(* CODESYS project festo_tcmc3.library
   Company: Festo AG & Co. KG
   DefaultNamespace: Festo_TcMC3
   Version: 3.1.1
   Placeholder: Festo TcMC Library for TwinCAT 3
   Author: Festo AG & Co. KG
   Title: Festo TcMC Library for TwinCAT 3
   Description: Additional Function blocks 
      to use Festo CMMx-xx Controller 
      with Beckhoff TwinCAT NC Environment

Project tree, tasks and I/O mapping:
  libraries: Tc2_EtherCAT, * (Beckhoff Automation GmbH); Tc2_Math, * (Beckhoff Automation GmbH); Tc2_MC2, * (Beckhoff Automation GmbH); Tc2_NC, * (Beckhoff Automation GmbH); Tc2_Standard, * (Beckhoff Automation GmbH); Tc2_System, * (Beckhoff Automation GmbH); Tc2_Utilities, * (Beckhoff Automation GmbH)
  Data types/
    data type EFesto_CAN_IDX
    data type EFesto_CAN_SUB_IDX
  POUs/
    function block Festo_GetDriveError [ST]
    function block Festo_MC_Home [ST]
    function block Festo_ReadCanObj [ST]
    function block Festo_WriteCanObj [ST]
  Version/
    global variables Global_Version
  Visualizations/
*)

// Data types/EFesto_CAN_IDX
TYPE EFesto_CAN_IDX :
(
	E_FESTO_CAN_IDX_NONE			:= 16#0,
	E_FESTO_CAN_IDX_ERROR			:= 16#1003

);
END_TYPE

// Data types/EFesto_CAN_SUB_IDX
TYPE EFesto_CAN_SUB_IDX :
(
	E_FESTO_CAN_IDX_SUB_00			:= 16#0,
	E_FESTO_CAN_IDX_SUB_01			:= 16#1,
	E_FESTO_CAN_IDX_SUB_02			:= 16#2,
	E_FESTO_CAN_IDX_SUB_03			:= 16#3,
	E_FESTO_CAN_IDX_SUB_04			:= 16#4,
	E_FESTO_CAN_IDX_SUB_05			:= 16#5,
	E_FESTO_CAN_IDX_SUB_06			:= 16#6,
	E_FESTO_CAN_IDX_SUB_07			:= 16#7,
	E_FESTO_CAN_IDX_SUB_08			:= 16#8,
	E_FESTO_CAN_IDX_SUB_09			:= 16#9,
	E_FESTO_CAN_IDX_SUB_0A			:= 16#0A,
	E_FESTO_CAN_IDX_SUB_0B			:= 16#0B,
	E_FESTO_CAN_IDX_SUB_0C			:= 16#0C,
	E_FESTO_CAN_IDX_SUB_0D			:= 16#0D,
	E_FESTO_CAN_IDX_SUB_0E			:= 16#0E,
	E_FESTO_CAN_IDX_SUB_0F			:= 16#0F,
	E_FESTO_CAN_IDX_SUB_10			:= 16#10,
	E_FESTO_CAN_IDX_SUB_11			:= 16#11,
	E_FESTO_CAN_IDX_SUB_12			:= 16#12,
	E_FESTO_CAN_IDX_SUB_13			:= 16#13,
	E_FESTO_CAN_IDX_SUB_14			:= 16#14,
	E_FESTO_CAN_IDX_SUB_15			:= 16#15,
	E_FESTO_CAN_IDX_SUB_16			:= 16#16,
	E_FESTO_CAN_IDX_SUB_17			:= 16#17,
	E_FESTO_CAN_IDX_SUB_18			:= 16#18,
	E_FESTO_CAN_IDX_SUB_19			:= 16#19,
	E_FESTO_CAN_IDX_SUB_1A			:= 16#1A,
	E_FESTO_CAN_IDX_SUB_1B			:= 16#1B,
	E_FESTO_CAN_IDX_SUB_1C			:= 16#1C,
	E_FESTO_CAN_IDX_SUB_1D			:= 16#1D,
	E_FESTO_CAN_IDX_SUB_1E			:= 16#1E,
	E_FESTO_CAN_IDX_SUB_1F			:= 16#1F,
	E_FESTO_CAN_IDX_SUB_20			:= 16#20,
	E_FESTO_CAN_IDX_SUB_21			:= 16#21,
	E_FESTO_CAN_IDX_SUB_22			:= 16#22,
	E_FESTO_CAN_IDX_SUB_23			:= 16#23,
	E_FESTO_CAN_IDX_SUB_24			:= 16#24,
	E_FESTO_CAN_IDX_SUB_25			:= 16#25,
	E_FESTO_CAN_IDX_SUB_26			:= 16#26,
	E_FESTO_CAN_IDX_SUB_27			:= 16#27,
	E_FESTO_CAN_IDX_SUB_28			:= 16#28,
	E_FESTO_CAN_IDX_SUB_29			:= 16#29,
	E_FESTO_CAN_IDX_SUB_2A			:= 16#2A,
	E_FESTO_CAN_IDX_SUB_2B			:= 16#2B,
	E_FESTO_CAN_IDX_SUB_2C			:= 16#2C,
	E_FESTO_CAN_IDX_SUB_2D			:= 16#2D,
	E_FESTO_CAN_IDX_SUB_2E			:= 16#2E,
	E_FESTO_CAN_IDX_SUB_2F			:= 16#2F,
	E_FESTO_CAN_IDX_SUB_30			:= 16#30,
	E_FESTO_CAN_IDX_SUB_31			:= 16#31,
	E_FESTO_CAN_IDX_SUB_32			:= 16#32,
	E_FESTO_CAN_IDX_SUB_33			:= 16#33,
	E_FESTO_CAN_IDX_SUB_34			:= 16#34,
	E_FESTO_CAN_IDX_SUB_35			:= 16#35,
	E_FESTO_CAN_IDX_SUB_36			:= 16#36,
	E_FESTO_CAN_IDX_SUB_37			:= 16#37,
	E_FESTO_CAN_IDX_SUB_38			:= 16#38,
	E_FESTO_CAN_IDX_SUB_39			:= 16#39,
	E_FESTO_CAN_IDX_SUB_3A			:= 16#3A,
	E_FESTO_CAN_IDX_SUB_3B			:= 16#3B,
	E_FESTO_CAN_IDX_SUB_3C			:= 16#3C,
	E_FESTO_CAN_IDX_SUB_3D			:= 16#3D,
	E_FESTO_CAN_IDX_SUB_3E			:= 16#3E,
	E_FESTO_CAN_IDX_SUB_3F			:= 16#3F,
	E_FESTO_CAN_IDX_SUB_40			:= 16#40,
	E_FESTO_CAN_IDX_SUB_41			:= 16#41,
	E_FESTO_CAN_IDX_SUB_42			:= 16#42,
	E_FESTO_CAN_IDX_SUB_43			:= 16#43,
	E_FESTO_CAN_IDX_SUB_44			:= 16#44,
	E_FESTO_CAN_IDX_SUB_45			:= 16#45,
	E_FESTO_CAN_IDX_SUB_46			:= 16#46,
	E_FESTO_CAN_IDX_SUB_47			:= 16#47,
	E_FESTO_CAN_IDX_SUB_48			:= 16#48,
	E_FESTO_CAN_IDX_SUB_49			:= 16#49,
	E_FESTO_CAN_IDX_SUB_4A			:= 16#4A,
	E_FESTO_CAN_IDX_SUB_4B			:= 16#4B,
	E_FESTO_CAN_IDX_SUB_4C			:= 16#4C,
	E_FESTO_CAN_IDX_SUB_4D			:= 16#4D,
	E_FESTO_CAN_IDX_SUB_4E			:= 16#4E,
	E_FESTO_CAN_IDX_SUB_4F			:= 16#4F,
	E_FESTO_CAN_IDX_SUB_50			:= 16#50,
	E_FESTO_CAN_IDX_SUB_51			:= 16#51,
	E_FESTO_CAN_IDX_SUB_52			:= 16#52,
	E_FESTO_CAN_IDX_SUB_53			:= 16#53,
	E_FESTO_CAN_IDX_SUB_54			:= 16#54,
	E_FESTO_CAN_IDX_SUB_55			:= 16#55,
	E_FESTO_CAN_IDX_SUB_56			:= 16#56,
	E_FESTO_CAN_IDX_SUB_57			:= 16#57,
	E_FESTO_CAN_IDX_SUB_58			:= 16#58,
	E_FESTO_CAN_IDX_SUB_59			:= 16#59,
	E_FESTO_CAN_IDX_SUB_5A			:= 16#5A,
	E_FESTO_CAN_IDX_SUB_5B			:= 16#5B,
	E_FESTO_CAN_IDX_SUB_5C			:= 16#5C,
	E_FESTO_CAN_IDX_SUB_5D			:= 16#5D,
	E_FESTO_CAN_IDX_SUB_5E			:= 16#5E,
	E_FESTO_CAN_IDX_SUB_5F			:= 16#5F,
	E_FESTO_CAN_IDX_SUB_60			:= 16#60,
	E_FESTO_CAN_IDX_SUB_61			:= 16#61,
	E_FESTO_CAN_IDX_SUB_62			:= 16#62,
	E_FESTO_CAN_IDX_SUB_63			:= 16#63,
	E_FESTO_CAN_IDX_SUB_64			:= 16#64,
	E_FESTO_CAN_IDX_SUB_65			:= 16#65,
	E_FESTO_CAN_IDX_SUB_66			:= 16#66,
	E_FESTO_CAN_IDX_SUB_67			:= 16#67,
	E_FESTO_CAN_IDX_SUB_68			:= 16#68,
	E_FESTO_CAN_IDX_SUB_69			:= 16#69,
	E_FESTO_CAN_IDX_SUB_6A			:= 16#6A,
	E_FESTO_CAN_IDX_SUB_6B			:= 16#6B,
	E_FESTO_CAN_IDX_SUB_6C			:= 16#6C,
	E_FESTO_CAN_IDX_SUB_6D			:= 16#6D,
	E_FESTO_CAN_IDX_SUB_6E			:= 16#6E,
	E_FESTO_CAN_IDX_SUB_6F			:= 16#6F,
	E_FESTO_CAN_IDX_SUB_70			:= 16#70,
	E_FESTO_CAN_IDX_SUB_71			:= 16#71,
	E_FESTO_CAN_IDX_SUB_72			:= 16#72,
	E_FESTO_CAN_IDX_SUB_73			:= 16#73,
	E_FESTO_CAN_IDX_SUB_74			:= 16#74,
	E_FESTO_CAN_IDX_SUB_75			:= 16#75,
	E_FESTO_CAN_IDX_SUB_76			:= 16#76,
	E_FESTO_CAN_IDX_SUB_77			:= 16#77,
	E_FESTO_CAN_IDX_SUB_78			:= 16#78,
	E_FESTO_CAN_IDX_SUB_79			:= 16#79,
	E_FESTO_CAN_IDX_SUB_7A			:= 16#7A,
	E_FESTO_CAN_IDX_SUB_7B			:= 16#7B,
	E_FESTO_CAN_IDX_SUB_7C			:= 16#7C,
	E_FESTO_CAN_IDX_SUB_7D			:= 16#7D,
	E_FESTO_CAN_IDX_SUB_7E			:= 16#7E,
	E_FESTO_CAN_IDX_SUB_7F			:= 16#7F,
	E_FESTO_CAN_IDX_SUB_80			:= 16#80,
	E_FESTO_CAN_IDX_SUB_81			:= 16#81,
	E_FESTO_CAN_IDX_SUB_82			:= 16#82,
	E_FESTO_CAN_IDX_SUB_83			:= 16#83,
	E_FESTO_CAN_IDX_SUB_84			:= 16#84,
	E_FESTO_CAN_IDX_SUB_85			:= 16#85,
	E_FESTO_CAN_IDX_SUB_86			:= 16#86,
	E_FESTO_CAN_IDX_SUB_87			:= 16#87,
	E_FESTO_CAN_IDX_SUB_88			:= 16#88,
	E_FESTO_CAN_IDX_SUB_89			:= 16#89,
	E_FESTO_CAN_IDX_SUB_8A			:= 16#8A,
	E_FESTO_CAN_IDX_SUB_8B			:= 16#8B,
	E_FESTO_CAN_IDX_SUB_8C			:= 16#8C,
	E_FESTO_CAN_IDX_SUB_8D			:= 16#8D,
	E_FESTO_CAN_IDX_SUB_8E			:= 16#8E,
	E_FESTO_CAN_IDX_SUB_8F			:= 16#8F,
	E_FESTO_CAN_IDX_SUB_90			:= 16#90,
	E_FESTO_CAN_IDX_SUB_91			:= 16#91,
	E_FESTO_CAN_IDX_SUB_92			:= 16#92,
	E_FESTO_CAN_IDX_SUB_93			:= 16#93,
	E_FESTO_CAN_IDX_SUB_94			:= 16#94,
	E_FESTO_CAN_IDX_SUB_95			:= 16#95,
	E_FESTO_CAN_IDX_SUB_96			:= 16#96,
	E_FESTO_CAN_IDX_SUB_97			:= 16#97,
	E_FESTO_CAN_IDX_SUB_98			:= 16#98,
	E_FESTO_CAN_IDX_SUB_99			:= 16#99,
	E_FESTO_CAN_IDX_SUB_9A			:= 16#9A,
	E_FESTO_CAN_IDX_SUB_9B			:= 16#9B,
	E_FESTO_CAN_IDX_SUB_9C			:= 16#9C,
	E_FESTO_CAN_IDX_SUB_9D			:= 16#9D,
	E_FESTO_CAN_IDX_SUB_9E			:= 16#9E,
	E_FESTO_CAN_IDX_SUB_9F			:= 16#9F,
	E_FESTO_CAN_IDX_SUB_A0			:= 16#A0,
	E_FESTO_CAN_IDX_SUB_A1			:= 16#A1,
	E_FESTO_CAN_IDX_SUB_A2			:= 16#A2,
	E_FESTO_CAN_IDX_SUB_A3			:= 16#A3,
	E_FESTO_CAN_IDX_SUB_A4			:= 16#A4,
	E_FESTO_CAN_IDX_SUB_A5			:= 16#A5,
	E_FESTO_CAN_IDX_SUB_A6			:= 16#A6,
	E_FESTO_CAN_IDX_SUB_A7			:= 16#A7,
	E_FESTO_CAN_IDX_SUB_A8			:= 16#A8,
	E_FESTO_CAN_IDX_SUB_A9			:= 16#A9,
	E_FESTO_CAN_IDX_SUB_AA			:= 16#AA,
	E_FESTO_CAN_IDX_SUB_AB			:= 16#AB,
	E_FESTO_CAN_IDX_SUB_AC			:= 16#AC,
	E_FESTO_CAN_IDX_SUB_AD			:= 16#AD,
	E_FESTO_CAN_IDX_SUB_AE			:= 16#AE,
	E_FESTO_CAN_IDX_SUB_AF			:= 16#AF,
	E_FESTO_CAN_IDX_SUB_B0			:= 16#B0,
	E_FESTO_CAN_IDX_SUB_B1			:= 16#B1,
	E_FESTO_CAN_IDX_SUB_B2			:= 16#B2,
	E_FESTO_CAN_IDX_SUB_B3			:= 16#B3,
	E_FESTO_CAN_IDX_SUB_B4			:= 16#B4,
	E_FESTO_CAN_IDX_SUB_B5			:= 16#B5,
	E_FESTO_CAN_IDX_SUB_B6			:= 16#B6,
	E_FESTO_CAN_IDX_SUB_B7			:= 16#B7,
	E_FESTO_CAN_IDX_SUB_B8			:= 16#B8,
	E_FESTO_CAN_IDX_SUB_B9			:= 16#B9,
	E_FESTO_CAN_IDX_SUB_BA			:= 16#BA,
	E_FESTO_CAN_IDX_SUB_BB			:= 16#BB,
	E_FESTO_CAN_IDX_SUB_BC			:= 16#BC,
	E_FESTO_CAN_IDX_SUB_BD			:= 16#BD,
	E_FESTO_CAN_IDX_SUB_BE			:= 16#BE,
	E_FESTO_CAN_IDX_SUB_BF			:= 16#BF,
	E_FESTO_CAN_IDX_SUB_C0			:= 16#C0,
	E_FESTO_CAN_IDX_SUB_C1			:= 16#C1,
	E_FESTO_CAN_IDX_SUB_C2			:= 16#C2,
	E_FESTO_CAN_IDX_SUB_C3			:= 16#C3,
	E_FESTO_CAN_IDX_SUB_C4			:= 16#C4,
	E_FESTO_CAN_IDX_SUB_C5			:= 16#C5,
	E_FESTO_CAN_IDX_SUB_C6			:= 16#C6,
	E_FESTO_CAN_IDX_SUB_C7			:= 16#C7,
	E_FESTO_CAN_IDX_SUB_C8			:= 16#C8,
	E_FESTO_CAN_IDX_SUB_C9			:= 16#C9,
	E_FESTO_CAN_IDX_SUB_CA			:= 16#CA,
	E_FESTO_CAN_IDX_SUB_CB			:= 16#CB,
	E_FESTO_CAN_IDX_SUB_CC			:= 16#CC,
	E_FESTO_CAN_IDX_SUB_CD			:= 16#CD,
	E_FESTO_CAN_IDX_SUB_CE			:= 16#CE,
	E_FESTO_CAN_IDX_SUB_CF			:= 16#CF,
	E_FESTO_CAN_IDX_SUB_D0			:= 16#D0,
	E_FESTO_CAN_IDX_SUB_D1			:= 16#D1,
	E_FESTO_CAN_IDX_SUB_D2			:= 16#D2,
	E_FESTO_CAN_IDX_SUB_D3			:= 16#D3,
	E_FESTO_CAN_IDX_SUB_D4			:= 16#D4,
	E_FESTO_CAN_IDX_SUB_D5			:= 16#D5,
	E_FESTO_CAN_IDX_SUB_D6			:= 16#D6,
	E_FESTO_CAN_IDX_SUB_D7			:= 16#D7,
	E_FESTO_CAN_IDX_SUB_D8			:= 16#D8,
	E_FESTO_CAN_IDX_SUB_D9			:= 16#D9,
	E_FESTO_CAN_IDX_SUB_DA			:= 16#DA,
	E_FESTO_CAN_IDX_SUB_DB			:= 16#DB,
	E_FESTO_CAN_IDX_SUB_DC			:= 16#DC,
	E_FESTO_CAN_IDX_SUB_DD			:= 16#DD,
	E_FESTO_CAN_IDX_SUB_DE			:= 16#DE,
	E_FESTO_CAN_IDX_SUB_DF			:= 16#DF,
	E_FESTO_CAN_IDX_SUB_E0			:= 16#E0,
	E_FESTO_CAN_IDX_SUB_E1			:= 16#E1,
	E_FESTO_CAN_IDX_SUB_E2			:= 16#E2,
	E_FESTO_CAN_IDX_SUB_E3			:= 16#E3,
	E_FESTO_CAN_IDX_SUB_E4			:= 16#E4,
	E_FESTO_CAN_IDX_SUB_E5			:= 16#E5,
	E_FESTO_CAN_IDX_SUB_E6			:= 16#E6,
	E_FESTO_CAN_IDX_SUB_E7			:= 16#E7,
	E_FESTO_CAN_IDX_SUB_E8			:= 16#E8,
	E_FESTO_CAN_IDX_SUB_E9			:= 16#E9,
	E_FESTO_CAN_IDX_SUB_EA			:= 16#EA,
	E_FESTO_CAN_IDX_SUB_EB			:= 16#EB,
	E_FESTO_CAN_IDX_SUB_EC			:= 16#EC,
	E_FESTO_CAN_IDX_SUB_ED			:= 16#ED,
	E_FESTO_CAN_IDX_SUB_EE			:= 16#EE,
	E_FESTO_CAN_IDX_SUB_EF			:= 16#EF,
	E_FESTO_CAN_IDX_SUB_F0			:= 16#F0,
	E_FESTO_CAN_IDX_SUB_F1			:= 16#F1,
	E_FESTO_CAN_IDX_SUB_F2			:= 16#F2,
	E_FESTO_CAN_IDX_SUB_F3			:= 16#F3,
	E_FESTO_CAN_IDX_SUB_F4			:= 16#F4,
	E_FESTO_CAN_IDX_SUB_F5			:= 16#F5,
	E_FESTO_CAN_IDX_SUB_F6			:= 16#F6,
	E_FESTO_CAN_IDX_SUB_F7			:= 16#F7,
	E_FESTO_CAN_IDX_SUB_F8			:= 16#F8,
	E_FESTO_CAN_IDX_SUB_F9			:= 16#F9,
	E_FESTO_CAN_IDX_SUB_FA			:= 16#FA,
	E_FESTO_CAN_IDX_SUB_FB			:= 16#FB,
	E_FESTO_CAN_IDX_SUB_FC			:= 16#FC,
	E_FESTO_CAN_IDX_SUB_FD			:= 16#FD,
	E_FESTO_CAN_IDX_SUB_FE			:= 16#FE,
	E_FESTO_CAN_IDX_SUB_FF			:= 16#FF
);
END_TYPE

// Version/Global_Version
// This function has been automatically generated from the project information.
VAR_GLOBAL CONSTANT
	{attribute 'const_non_replaced'}
	stLibVersion_Festo_TcMC_Library_for_TwinCAT_3 : ST_LibVersion := (iMajor := 3, iMinor := 1, iBuild := 1, iRevision := 0, sVersion := '3.1.1');
END_VAR

// POUs/Festo_GetDriveError
(****************************************************************************************************************
     FESTO AG  Co., Esslingen                                                    								
     Copyright (c) 2014. All rights reserved.                       

 Functionblock:  Festo_GetDriveError
 Description:    Function block for CMMx-xx
				 If there is an Error on the NC-StatusWord, the function starts reading Error 1-4 from the Drive
				 The function communicates via SDO with the Drive

 Version:        V2.0        
 Composer:       bejk
 Date:           02.01.2014                                                                           
****************************************************************************************************************)
{library private}
(****************************************************************************************************************
Date          Name                      Activity                                                                              
                                                            
11.11.2011    Benjamin Kilgus           created
02.01.2014    Daniel Heihsel            SDO Reading via seperate functions; get ErrorArray[0..3], no stringoutput
****************************************************************************************************************)
{library public}
FUNCTION_BLOCK Festo_GetDriveError
VAR_INPUT
	DeviceType                  	: USINT:=0; 				(* DeviceTye: 0 = Coe - EtherCat, 1 = CanOpen *)
	Enable                   	    : BOOL;
	DeviceNetID                 	: T_AmsNetId;
	DevicePort                  	: T_AmsPort;
	ErrorPullTime					: TIME := t#500ms;
	NCStateDWord					: DWORD; 					(* StateDWord from NcToPlc-structure *)
END_VAR
VAR_OUTPUT
	Busy                        	: BOOL;
	DriveInErrorState           	: BOOL;	    				(* Drive in error State *)
	DriveErrorNumber    	        : ARRAY [1..4] OF DWORD;  	(* Number of actual Error *)
	Error                       	: BOOL;	     				(* Error flag *)
	ErrorId                     	: UDINT;	     			(* Error code *)
END_VAR

VAR
	ReadCANobject              		: Festo_ReadCanObj;
	ADSTimeOut   		  	      	: TIME := DEFAULT_ADS_TIMEOUT;
	tonWait							: TON;
	State							: INT;
	IndexCounter					: INT;
	IndexCounterMax 				: INT;

	DriveErrorNumberClear     	  	: ARRAY [1..4] OF DWORD;  (* Number of actual Error *)
	DriveInErrorStateLast			: BOOL;
END_VAR

(* Map Status ErrorBit *)
DriveInErrorState := AxisDriveDeviceError(NCStateDWord) AND Enable;

(* delete ErrorArray
 -> switch Enable on OR Drive switch in ErrorState *)
	IF DriveInErrorState
	AND NOT  DriveInErrorStateLast
	THEN
		DriveErrorNumber := DriveErrorNumberClear;
	ELSIF DriveInErrorState
	AND NOT  DriveInErrorStateLast
	THEN
		DriveErrorNumber := DriveErrorNumberClear;
	END_IF

(* Read immediatly last error with ErrorBit *)
ReadCANobject(
					Execute			:= ,
					DeviceType		:= DeviceType,	(* DeviceTye: 0 = Coe - EtherCat, 1 = CanOpen *)
					DeviceNetID		:= DeviceNetID,
					DevicePort		:= DevicePort,
					Index			:= E_FESTO_CAN_IDX_ERROR,
					SubIndex		:= ,
					DestAddr		:= ,
					DataLength		:= SIZEOF(DriveErrorNumber[1]),
					ADSTimeOut	 	:= ,
					Busy			=> ,
					Error			=> Error,
					ErrorId			=> ErrorId
					);


CASE State OF
0:
	IF Enable THEN
		Busy := TRUE;
		State := 10;
		IndexCounter := 1;
		IndexCounterMax := SIZEOF(DriveErrorNumber)/SIZEOF(DriveErrorNumber[1]);
	ELSE
		Busy := FALSE;
	END_IF
10:
	IF NOT Enable THEN
		State := 0;
		Busy := FALSE;
	ELSIF DriveInErrorState THEN
		ReadCANobject(Execute := FALSE);
		IndexCounter := 1;
		State := 11;
	END_IF

11:
	ReadCANobject.SubIndex			:= INT_TO_BYTE(E_FESTO_CAN_IDX_SUB_00 + IndexCounter);
	ReadCANobject.DestAddr			:= ADR(DriveErrorNumber[IndexCounter]);
	ReadCANobject(Execute := TRUE);
	State := 12;

12:
	IF NOT ReadCANobject.Busy
	THEN
		IF ReadCANobject.Error THEN
				ErrorId := ReadCANobject.ErrorId;
				State := 20;
		ELSE
			IF IndexCounter < IndexCounterMax THEN
				IndexCounter := IndexCounter + 1;
				State := 11;
			ELSE
				IndexCounter := 1;
				State := 20;
			END_IF
		END_IF
		ReadCANobject(Execute := FALSE);
	END_IF

20:
	tonWait(IN := TRUE, PT := ErrorPullTime);
	IF tonWait.Q THEN
		tonWait(IN := FALSE);
		State := 10;
	ELSIF NOT DriveInErrorState THEN
		tonWait(IN := FALSE);
		State := 10;
	END_IF

(* ERROR-STATE *)
900:
	Error := TRUE;
	IF NOT Enable THEN
		State := 0;
	END_IF

END_CASE

(* Save actual Value for next cycle *)
DriveInErrorStateLast  := DriveInErrorState;

END_FUNCTION_BLOCK

// POUs/Festo_ReadCanObj
FUNCTION_BLOCK Festo_ReadCanObj
(****************************************************************************************************************
     FESTO AG  Co., Esslingen                                                    								
     Copyright (c) 2011. All rights reserved.                       

 Functionblock:	Festo_ReadCanObj
 Description:	Function block for CMMx-xx
				Reads the CANOpen- / CoE-Object via SDO

 Version:        V2.0        
 Composer:       heihdan
 Date:           10.12.2013                                                                           
****************************************************************************************************************)
{library private}
(****************************************************************************************************************
Date          Name                      Activity                                                                              
                                                            
10.12.2013    Daniel Heihsel			created
17.05.2016    Christian Hammer			changed datatype for DestAddr from UDINT to PVOID
****************************************************************************************************************)
{library public}
VAR_INPUT
	Execute			: BOOL;
	DeviceType		: USINT;	(* DeviceTye: 0 = Coe - EtherCat, 1 = CanOpen *)
	DeviceNetID		: T_AmsNetId;
	DevicePort		: T_AmsPort;
	Index			: WORD;
	SubIndex		: BYTE;
	DestAddr		: PVOID;
	DataLength		: UDINT;
	ADSTimeOut 		: TIME := DEFAULT_ADS_TIMEOUT;
END_VAR
VAR_OUTPUT
	Busy			: BOOL;
	Error			: BOOL;
	ErrorId			: UDINT;
END_VAR
VAR
	ReadCANobject	: ADSREAD;
	FB_ADSEcCoREAD	: FB_EcCoESdoRead;
END_VAR

	(* CANopen DEVICE *)
IF DeviceType = 1 THEN
	ReadCANobject(
		READ            := Execute,
		NETID           := DeviceNetID,
		PORT            := DevicePort,
		IDXGRP          := Index,
		IDXOFFS         := SubIndex,
		DESTADDR        := DestAddr,
		LEN				:= DataLength,
		TMOUT           := ADSTimeOut,
		BUSY            => Busy,
		ERR             => Error,
		ERRID           => ErrorId);

(* EtherCAT DEVICE *)
ELSE
  FB_ADSEcCoREAD(
    bExecute   			:= Execute,
	sNetId     			:= DeviceNetID,
    nSlaveAddr 			:= DevicePort,
    nIndex     			:= Index,
    nSubIndex  			:= SubIndex,
    pDstBuf    			:= DestAddr,
    cbBufLen   			:= DataLength,
    tTimeout   			:= ADSTimeOut,
    bBusy      			=> Busy,
    bError    		 	=> Error,
    nErrId     			=> ErrorId);
END_IF;

END_FUNCTION_BLOCK

// POUs/Festo_MC_Home
(****************************************************************************************************************
     FESTO AG  Co., Esslingen                                                    								
     Copyright (c) 2014. All rights reserved.                       

 Functionblock:  Festo_MC_Home
 Description:    Funktion block for CMMx-xx (Beckhoff TcMC2.lib)
 Version:        V1.1        
 Composer:       bejk
 Date:           10.11.2011                                                                           
****************************************************************************************************************)

(****************************************************************************************************************
Date          	Name	Activity                                                                              
                                                            
10.11.2011    	bejk	created
10.07.2014		bejk	geänderte Bedingung für Fehler Referenzfahrt step 50 (DriveStateWord.3) 
****************************************************************************************************************)
{library public}
FUNCTION_BLOCK Festo_MC_Home
VAR_INPUT
	DeviceType                  :USINT:=0;
(* 0 -> CMx-xx EtherCAT
   1 -> CMx-xx CANopen  *)
	Execute                     :BOOL;  (* start execution *)
	DeviceNetID                 :T_AmsNetId;
	DevicePort                  :UINT;
END_VAR
VAR_OUTPUT
	Done                        :BOOL;	(* successfully done *)
	CommandAborted              :BOOL;	(* aborted *)
	Busy                        :BOOL;	(* busy, not in initial state *)
	Error                       :BOOL;	(* Error flag *)
	ErrorId                     :UDINT;	(* Error code *)
END_VAR

VAR_IN_OUT
	Axis                        :AXIS_REF;
END_VAR
{library private}
VAR
	abort                       :BOOL;
	bRead                       :BOOL;
	bWrite                      :BOOL;
	bReadDone                   :BOOL;
	bWriteDone                  :BOOL;
	bError                      :BOOL;
	DriveOPMDisplay             :UINT;
	LagDistanceMonitoring       :UINT;
	SavedLagDistanceMonitoring  :UINT;
	state                       :INT;
	ErrorState                  :INT;
	IdxGroup                    :WORD;
	IdxOffs                     :BYTE;
	Length                      :UDINT;
	Buffer                      :DWORD;
    Const_StartMode             :INT   :=16#F;
    Const_HomingMode            :USINT :=6;
    Const_IPMode                :USINT :=7;
	Const_CearBuffer            :USINT :=1;
	DriveStateWord              :WORD;
	NcReferenceFlag             :DWORD;
	tADSTimeOut   		        :TIME  :=T#1s;
	WriteCANobject              :ADSWRITE;
	ReadCANobject               :ADSREAD;
	FB_ADSEcCoWRITE             :FB_EcCoESdoWrite;
	FB_ADSEcCoREAD              :FB_EcCoESdoRead;
	WriteNC                     :ADSWRITE;
	ReadNC                      :ADSREAD;
	Timeout                     :TON;
	ExecuteOnTrigger            :R_TRIG;
	ExecuteOffTrigger           :F_TRIG;
	SetActualPosition           :MC_SetPosition;
END_VAR
{library public}

ExecuteOffTrigger(CLK:=Execute);

  bWriteDone   := FALSE;
  bReadDone    := FALSE;
  bError       := FALSE;

(* CANopen DEVICE *)
IF DeviceType = 1 THEN
  WriteCANobject(
    NETID            := DeviceNetID,
    PORT             := DevicePort,
    IDXGRP           := IdxGroup,
    IDXOFFS          := IdxOffs,
    LEN              := Length,
 	SRCADDR          := ADR(Buffer),
	WRITE            := bWrite,
	TMOUT            := tADSTimeOut,
	BUSY             => ,
	ERR              => ,
	ERRID            => );

ReadCANobject(
    NETID            := DeviceNetID,
    PORT             := DevicePort,
    IDXGRP           := IdxGroup,
    IDXOFFS          := IdxOffs,
    LEN              := Length,
	DESTADDR         := ADR(Buffer),
	READ             := bRead,
	TMOUT            := tADSTimeOut,
	BUSY             => ,
	ERR              => ,
	ERRID            => );

  IF bWrite THEN
    IF NOT ReadCANobject.BUSY AND NOT ReadCANobject.ERR THEN
      bWriteDone    := TRUE;
    ELSIF NOT ReadCANobject.BUSY AND ReadCANobject.ERR THEN
      bError        := TRUE;
      abort         := TRUE;
      ErrorId       := ReadCANobject.ERRID;
      ErrorState    := state;
      state         := 1020;
	END_IF;
  END_IF

  IF bRead THEN
    IF NOT ReadCANobject.BUSY AND NOT ReadCANobject.ERR THEN
      bReadDone     := TRUE;
    ELSIF NOT ReadCANobject.BUSY AND ReadCANobject.ERR THEN
      bError        := TRUE;
      abort         := TRUE;
      ErrorId       := ReadCANobject.ERRID;
      ErrorState    := state;
      state         := 1020;
	END_IF;
END_IF;

(* EtherCAT DEVICE *)
ELSE
  FB_ADSEcCoWRITE(
    sNetId     := DeviceNetID,
    nSlaveAddr := DevicePort,
    nSubIndex  := IdxOffs,
    nIndex     := IdxGroup,
    pSrcBuf    := ADR(Buffer),
    cbBufLen   := Length,
    bExecute   := bWrite,
    tTimeout   := tADSTimeOut,
    bBusy      => ,
    bError     => ,
    nErrId     => );

  FB_ADSEcCoREAD(
    sNetId     := DeviceNetID,
    nSlaveAddr := DevicePort,
    nSubIndex  := IdxOffs,
    nIndex     := IdxGroup,
    pDstBuf    := ADR(Buffer),
    cbBufLen   := Length,
    bExecute   := bRead,
    tTimeout   := tADSTimeOut,
    bBusy      => ,
    bError     => ,
    nErrId     => );

  IF bRead THEN
    IF NOT FB_ADSEcCoREAD.bBusy AND NOT FB_ADSEcCoREAD.bError THEN
      bReadDone     := TRUE;
    ELSIF NOT FB_ADSEcCoREAD.bBusy AND FB_ADSEcCoREAD.bError THEN
      bError        := TRUE;
      abort         := TRUE;
      ErrorId       := FB_ADSEcCoREAD.nErrId;
      ErrorState    := state;
      state         := 1020;
    END_IF;
  END_IF;

  IF bWrite THEN
    IF NOT FB_ADSEcCoWRITE.bBusy AND NOT FB_ADSEcCoWRITE.bError THEN
      bwriteDone    := TRUE;
    ELSIF NOT FB_ADSEcCoWRITE.bBusy AND FB_ADSEcCoWRITE.bError THEN
      bError        := TRUE;
      abort         := TRUE;
      ErrorId       := FB_ADSEcCoWRITE.nErrId;
      ErrorState    := state;
      state         := 1020;
    END_IF;
  END_IF;
END_IF;

CASE state OF
	0 : (* initial state, wait for trigger *)
    	Busy                  := FALSE;
		Done                  := FALSE;
        abort                 := FALSE;
		CommandAborted        := FALSE;
		Error                 := FALSE;
		ErrorID               := 0;
		ErrorState            := 0;
        bRead                 := FALSE;
        bWrite                := FALSE;
		Timeout               ( IN      :=FALSE);
		ExecuteOnTrigger      ( CLK     :=Execute );

		IF ExecuteOnTrigger.Q THEN
          Busy                := TRUE;
          state               := 1;
		END_IF

     1: (* Check Stateword *)
    (* drive is operational and not moving *)
    IF Axis.NcToPlc.StateDWord.0 AND Axis.NcToPlc.StateDWord.2 THEN
      state         := 10;
    ELSE
      abort         := TRUE;
      ErrorId       := 16#FFFFFFF0;	(* Device not ready *);
      ErrorState    := state;
      state         := 1020;
    END_IF;

	10 : (* set opm to 6 (Homing Methode)*)
	  IdxGroup             := 16#6060;
	  IdxOffs              := 0;
	  Length               := SIZEOF(Const_HomingMode);
	  Buffer               := Const_HomingMode;
      bWrite               := TRUE;
      IF bWriteDone THEN
        bWrite             := FALSE;
	    state              := 20;
      END_IF;

	20 : (* read lag distance monitoring parameter *)
		ReadNC(NETID:='' , PORT:=AMSPORT_R0_NC , IDXGRP:=NCIDXG_AXPARMS+DWORD_TO_UINT(Axis.NcToPlc.AxisId) , IDXOFFS:=16#20010 , LEN:=SIZEOF(SavedLagDistanceMonitoring) , DESTADDR:=ADR(SavedLagDistanceMonitoring) , READ:=TRUE , TMOUT:=tADSTimeOut);
		IF NOT ReadNC.Busy AND NOT ReadNC.Err THEN
          ReadNC( READ:=FALSE );
          state         := 30;
		END_IF

	30 : (* disable lag distance monitoring *)
		LagDistanceMonitoring := 0;
		WriteNC(NETID:='' , PORT:=AMSPORT_R0_NC , IDXGRP:=NCIDXG_AXPARMS+DWORD_TO_UINT(Axis.NcToPlc.AxisId) , IDXOFFS:=16#20010 , LEN:=SIZEOF(LagDistanceMonitoring) , SRCADDR:=ADR(LagDistanceMonitoring) , WRITE:=TRUE , TMOUT:=T#1s);
		IF NOT WriteNC.Busy AND NOT WriteNC.Err THEN
          WriteNC( WRITE:=FALSE );
          state         := 35;
		END_IF

	35 : (* disable NC reference flag *)
		NcReferenceFlag := 0;
		WriteNC(NETID:='' , PORT:=AMSPORT_R0_NC , IDXGRP:=NCIDXG_AXFUNCS+DWORD_TO_UINT(Axis.NcToPlc.AxisId) , IDXOFFS:=16#1B , LEN:=SIZEOF(NcReferenceFlag) , SRCADDR:=ADR(NcReferenceFlag) , WRITE:=TRUE , TMOUT:=T#1s);
		IF NOT WriteNC.Busy AND NOT WriteNC.Err THEN
          WriteNC( WRITE:=FALSE );
          state         := 40;
		END_IF

	40 : (* Start Homing run via SDO *)
	  IdxGroup             := 16#6040;
	  IdxOffs              := 0;
	  Length               := SIZEOF(Const_StartMode);
	  Buffer               := Const_StartMode;
      bWrite               := TRUE;
      IF bWriteDone THEN
        bWrite             := FALSE;
	    state              := 50;
      END_IF;

	50 : (* wait Homing run to be done *)
	  IdxGroup             := 16#6041;
	  IdxOffs              := 0;
	  Length               := SIZEOF(DriveStateWord);
      bRead                := TRUE;
      IF bReadDone THEN
      bRead                := FALSE;
        DriveStateWord     := DWORD_TO_WORD(Buffer);
        IF DriveStateWord.12 THEN
          state            := 60;
          (* ref error *)
        ELSIF DriveStateWord.3 THEN
            Error          := TRUE;
            ErrorID        := 16#FFFFFFFE;	(* Homing ended with error *)
            ErrorState     := state;
            state          := 999;
          END_IF;
      END_IF;

	60 : (* set TwinCAT NC axis position to HomePosition value *)
        SetActualPosition(
	      Execute     := TRUE,
	      Position    := Axis.NcToPlc.ActPos,
          Mode        := ,
	      Options     := ,
	      Axis        := Axis,
	      Done        => ,
	      Busy        => ,
	      Error       => ,
	      ErrorID     => );
         SetActualPosition.Options.ClearPositionLag := TRUE;
		IF SetActualPosition.Done AND NOT SetActualPosition.Error THEN
			SetActualPosition(Execute:=FALSE, Axis:=Axis);
		    state        := 70;
        ELSIF SetActualPosition.Error THEN
            SetActualPosition(Execute:=FALSE, Axis:=Axis);
		    ErrorState   := state;
            state        := 999;
		END_IF

	70 : (* set opm to 7 (IP Mode)*)
	  IdxGroup             := 16#6060;
	  IdxOffs              := 0;
	  Length               := SIZEOF(Const_IPMode);
	  Buffer               := Const_IPMode;
      bWrite               := TRUE;
      IF bWriteDone THEN
        bWrite             := FALSE;
	    state              := 80;
      END_IF;

	80 : (* wait for OPMDisplay = 7  *)
	  IdxGroup             := 16#6061;
	  IdxOffs              := 0;
	  Length               := SIZEOF(DriveOPMDisplay);
      bRead                := TRUE;
      Timeout(IN:=TRUE , PT:=t#5000ms );
      IF bReadDone THEN
        bRead              := FALSE;
        DriveOPMDisplay    := DWORD_TO_UINT(Buffer);
        IF DriveOPMDisplay = 7 THEN
          Timeout.IN       := FALSE;
          state            := 90;
        (* not ok *)
        ELSIF Timeout.Q THEN
          Timeout.IN       := FALSE;
          ErrorState       := state;
          state            := 1010;
        END_IF;
      END_IF;

	90 : (* start Ip Mode *)
	  IdxGroup             := 16#6040;
	  IdxOffs              := 0;
	  Length               := SIZEOF(Const_StartMode);
	  Buffer               := Const_StartMode;
      bWrite               := TRUE;
      IF bWriteDone THEN
        bWrite             := FALSE;
	    state              := 100;
      END_IF;

	100 : (* set lag distance monitoring to its original value *)
		WriteNC(NETID:='' , PORT:=AMSPORT_R0_NC , IDXGRP:=NCIDXG_AXPARMS+DWORD_TO_UINT(Axis.NcToPlc.AxisId) , IDXOFFS:=16#20010 , LEN:=SIZEOF(SavedLagDistanceMonitoring) , SRCADDR:=ADR(SavedLagDistanceMonitoring) , WRITE:=TRUE , TMOUT:=T#1s);
		IF NOT WriteNC.Busy AND NOT WriteNC.ERR THEN
			WriteNC( WRITE:=FALSE );
			state := 110;
		END_IF

	110 : (* Enable NC reference flag *)
		NcReferenceFlag := 1;
		WriteNC(NETID:='' , PORT:=AMSPORT_R0_NC , IDXGRP:=NCIDXG_AXFUNCS+DWORD_TO_UINT(Axis.NcToPlc.AxisId) , IDXOFFS:=16#1B , LEN:=SIZEOF(NcReferenceFlag) , SRCADDR:=ADR(NcReferenceFlag) , WRITE:=TRUE , TMOUT:=T#1s);
		IF NOT WriteNC.Busy AND NOT WriteNC.ERR THEN
			WriteNC( WRITE:=FALSE );
			state := 120;
		END_IF

     120: (* finished *)
		Busy   := FALSE;
		Done   := TRUE;
        IF NOT Execute THEN
          state := 0;
        END_IF;

	(*============= ABORT =================*)

	999 : (* set opm to 7 (IP Mode) when Homing run ended with error *)
	  IdxGroup             := 16#6060;
	  IdxOffs              := 0;
	  Length               := SIZEOF(Const_IPMode);
	  Buffer               := Const_IPMode;
      bWrite               := TRUE;
      IF bWriteDone THEN
        bWrite             := FALSE;
	    state              := 1000;
      END_IF;

	1000 : (* wait for OPMDisplay = 7  *)
	  IdxGroup             := 16#6061;
	  IdxOffs              := 0;
	  Length               := SIZEOF(DriveOPMDisplay);
      bRead                := TRUE;
      Timeout(IN:=TRUE , PT:=t#5000ms );
      IF bReadDone THEN
        bRead              := FALSE;
        DriveOPMDisplay    := DWORD_TO_UINT(Buffer);
        IF DriveOPMDisplay = 7 THEN
          Timeout.IN       := FALSE;
          state            := 1010;
        (* not ok *)
        ELSIF Timeout.Q THEN
          Timeout.IN       := FALSE;
          ErrorState       := state;
          state            := 1020;
        END_IF;
      END_IF;


	1010: (* set lag distance monitoring to its original value *)
		LagDistanceMonitoring := 0;
		WriteNC(NETID:='' , PORT:=AMSPORT_R0_NC , IDXGRP:=NCIDXG_AXPARMS+DWORD_TO_UINT(Axis.NcToPlc.AxisId) , IDXOFFS:=16#20010 , LEN:=SIZEOF(SavedLagDistanceMonitoring) , SRCADDR:=ADR(SavedLagDistanceMonitoring) , WRITE:=TRUE , TMOUT:=T#1s);
		IF NOT WriteNC.Busy AND NOT WriteNC.ERR THEN
			WriteNC( WRITE:=FALSE );
			state := 1020;
		END_IF

     1020: (* finished with error *)
		Busy             := FALSE;
        Error            := TRUE;
        CommandAborted   := abort;
        IF NOT Execute THEN
          state          := 0;
        END_IF;
END_CASE;

END_FUNCTION_BLOCK

// POUs/Festo_WriteCanObj
FUNCTION_BLOCK Festo_WriteCanObj
(****************************************************************************************************************
     FESTO AG  Co., Esslingen                                                    								
     Copyright (c) 2011. All rights reserved.                       

 Functionblock:	Festo_ReadCanObj
 Description:	Function block for CMMx-xx
				Writes the CANOpen- / CoE-Object via SDO

 Version:        V2.0        
 Composer:       heihdan
 Date:           10.12.2013                                                                           
****************************************************************************************************************)
{library private}
(****************************************************************************************************************
Date          Name                      Activity                                                                              
                                                            
10.12.2013    Daniel Heihsel			created
17.05.2016    Christian Hammer			changed datatype for SrcAddr from UDINT to PVOID
****************************************************************************************************************)
{library public}
VAR_INPUT
	Execute			: BOOL;
	DeviceType		: USINT;	(* DeviceTye: 0 = Coe - EtherCat, 1 = CanOpen *)
	DeviceNetID		: T_AmsNetId;
	DevicePort		: T_AmsPort;
	Index			: WORD;
	SubIndex		: BYTE;
	SrcAddr			: PVOID;
	DataLength		: UDINT;
	ADSTimeOut		: TIME := DEFAULT_ADS_TIMEOUT;
END_VAR
VAR_OUTPUT
	Busy			: BOOL;
	Error			: BOOL;
	ErrorId			: UDINT;
END_VAR
VAR
	WriteCANobject	: ADSWRITE;
	FB_ADSEcCoWRITE	: FB_EcCoESdoWrite;
END_VAR

(* CANopen DEVICE *)
IF DeviceType = 1 THEN
	WriteCANobject(
		WRITE           := Execute,
		NETID           := DeviceNetID,
    	PORT            := DevicePort,
   		IDXGRP          := Index,
    	IDXOFFS         := SubIndex,
		SRCADDR         :=	SrcAddr,
		LEN				:= DataLength,
		TMOUT           := ADSTimeOut,
		BUSY            => Busy,
		ERR             => Error,
		ERRID           => ErrorId);

(* EtherCAT DEVICE *)
ELSE
  FB_ADSEcCoWRITE(
    bExecute   			:= Execute,
	sNetId     			:= DeviceNetID,
    nSlaveAddr 			:= DevicePort,
    nIndex     			:= Index,
    nSubIndex  			:= SubIndex,
    pSrcBuf    			:= SrcAddr,
    cbBufLen   			:= DataLength,
    tTimeout   			:= ADSTimeOut,
    bBusy      			=> Busy,
    bError    		 	=> Error,
    nErrId     			=> ErrorId);
END_IF;

END_FUNCTION_BLOCK
